TYPE T_CAC_Filename : T_MaxString;
END_TYPE

(* stored: Version 1.1.0.1
   DUT T_CAC_Filename: Id {18b6fa6e-75c5-480e-80a6-813af4e72ac2} *)
